FUNCTION_BLOCK Discrete_PI_LREAL3 (* Composite Function Block Type *)
  (* Standard: 61499-2 *)
  (* Version 0.0, 2018-07-31, 4DIAC-IDE, 4DIAC-Consortium *)
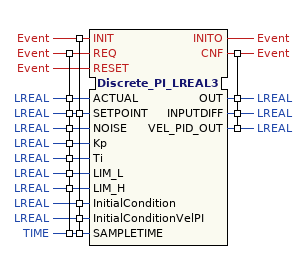
  EVENT_INPUT
    INIT WITH SAMPLETIME, SETPOINT, InitialCondition, InitialConditionVelPI; (* Initialization Request *)
    REQ WITH SAMPLETIME, ACTUAL, SETPOINT, NOISE, Kp, Ti, LIM_L, LIM_H; (* Normal Execution Request *)
    RESET;
  END_EVENT
  EVENT_OUTPUT
    INITO; (* Initialization Confirm *)
    CNF WITH OUT, INPUTDIFF, VEL_PID_OUT; (* Execution Confirmation *)
  END_EVENT
  VAR_INPUT
    ACTUAL : LREAL;
    SETPOINT : LREAL;
    NOISE : LREAL;
    Kp : LREAL;
    Ti : LREAL;
    LIM_L : LREAL;
    LIM_H : LREAL;
    InitialCondition : LREAL;
    InitialConditionVelPI : LREAL;
    SAMPLETIME : TIME;
  END_VAR
  VAR_OUTPUT
    OUT : LREAL;
    INPUTDIFF : LREAL;
    VEL_PID_OUT : LREAL;
  END_VAR
  FBS
    F_ADD : F_ADD;
    F_FT_LIMIT : F_FT_LIMIT;
    Delay_With_InitCondition : Delay_With_InitCondition;
    F_REAL_TO_LREAL : F_REAL_TO_LREAL;
    F_LREAL_TO_REAL : F_LREAL_TO_REAL;
    LIM_H : F_LREAL_TO_REAL;
    LIM_L : F_LREAL_TO_REAL;
    Velocity_PI_LREAL3 : Velocity_PI_LREAL3;
  END_FBS
  EVENT_CONNECTIONS
    REQ TO Delay_With_InitCondition.Start_and_REQ;
    F_REAL_TO_LREAL.CNF TO Delay_With_InitCondition.Start_and_REQ;
    F_FT_LIMIT.CNF TO F_REAL_TO_LREAL.REQ;
    Delay_With_InitCondition.CNF TO CNF;
    F_LREAL_TO_REAL.CNF TO F_FT_LIMIT.REQ;
    F_ADD.CNF TO F_LREAL_TO_REAL.REQ;
    REQ TO LIM_H.REQ;
    LIM_H.CNF TO F_FT_LIMIT.REQ;
    REQ TO LIM_L.REQ;
    LIM_L.CNF TO F_FT_LIMIT.REQ;
    INIT TO Velocity_PI_LREAL3.INIT;
    REQ TO Velocity_PI_LREAL3.REQ;
    RESET TO Velocity_PI_LREAL3.RESET;
    Velocity_PI_LREAL3.INITO TO Delay_With_InitCondition.INIT;
    Velocity_PI_LREAL3.INITO TO INITO;
    Velocity_PI_LREAL3.CNF TO F_ADD.REQ;
    Velocity_PI_LREAL3.CNF TO CNF;
    Delay_With_InitCondition.CNF TO F_ADD.REQ;
  END_CONNECTIONS
  DATA_CONNECTIONS
    SAMPLETIME TO Delay_With_InitCondition.DelayTime;
    F_FT_LIMIT.OUT TO F_REAL_TO_LREAL.IN;
    F_REAL_TO_LREAL.OUT TO Delay_With_InitCondition.DelayedInput;
    F_LREAL_TO_REAL.OUT TO F_FT_LIMIT.VAL;
    F_ADD.OUT TO F_LREAL_TO_REAL.IN;
    InitialCondition TO Delay_With_InitCondition.InitialCondition;
    LIM_H TO LIM_H.IN;
    LIM_H.OUT TO F_FT_LIMIT.LIM_H;
    LIM_L.OUT TO F_FT_LIMIT.LIM_L;
    LIM_L TO LIM_L.IN;
    ACTUAL TO Velocity_PI_LREAL3.ACTUAL;
    SETPOINT TO Velocity_PI_LREAL3.SETPOINT;
    NOISE TO Velocity_PI_LREAL3.NOISE;
    Kp TO Velocity_PI_LREAL3.KP;
    Ti TO Velocity_PI_LREAL3.Ti;
    InitialConditionVelPI TO Velocity_PI_LREAL3.InitialCondition;
    SAMPLETIME TO Velocity_PI_LREAL3.SAMPLETIME_ECYCLE;
    Velocity_PI_LREAL3.INPUTDIFF TO INPUTDIFF;
    Velocity_PI_LREAL3.DELTAOUTPUT TO F_ADD.IN1;
    Velocity_PI_LREAL3.DELTAOUTPUT TO VEL_PID_OUT;
    Delay_With_InitCondition.LREAL1 TO OUT;
    Delay_With_InitCondition.LREAL1 TO F_ADD.IN2;
  END_CONNECTIONS
END_FUNCTION_BLOCK
